Staubli VAL3: deb.pgx

program deb()
begin

end
